TEXTLIST TextList_Config_IAD
  0 = 'Config IAD' | FR: 'Configuration IAD' | EN: 'IAD Configuration'
  1 = 'Seuil ala' | FR: "Seuil d'alarme" | EN: 'Alarm threshold'
  2 = 'Temps av ala' | FR: 'Temps avant alarme' | EN: 'Delay before alarm'
  3 = 'Seuil def' | FR: 'Seuil de défaut' | EN: 'Default threshold'
  4 = 'Temps av def' | FR: 'Temps avant défaut' | EN: 'Delay before fault'
  5 = 'Tension anode' | FR: "Tension d'anode" | EN: 'Anode voltage'
  6 = 'Courant anode' | FR: "Courant d'anode" | EN: 'Anode current'
  7 = 'Courant neut' | FR: 'Courant neutraliseur' | EN: 'Neutralization current'
   = ''
END_TEXTLIST

(* stored: Version 1.1.0.1, ProductVersion 3.1.4024.10
   TextList TextList_Config_IAD: Id {73e3e62e-ea9d-4ab8-bc8c-0eac0882a323} *)
